{attribute 'linkalways'} 
{attribute 'no_explicit_call' := 'This FB is a CLASS and must be accessed using methods or properties'}
{attribute 'enable_dynamic_creation'}
FUNCTION_BLOCK _ETcVnVectorCompareMethod EXTENDS EnumDatatypeBase
VAR
	localData : ETcVnVectorCompareMethod;
	activeData : REFERENCE TO ETcVnVectorCompareMethod;
	enumBaseDatatype : _DINT(localData);
END_VAR

METHOD PRIVATE AddLocalEnumeration
VAR_INPUT
	Enumeration : T_MAXSTRING;
	Value : ETcVnVectorCompareMethod;
END_VAR
AddEnumeration(Enumeration, Value);
END_METHOD

PROPERTY PUBLIC Address : PVOID
GET
Address := ADR(activeData);
END_GET
END_PROPERTY

METHOD PUBLIC ClearReference
VAR_INPUT
END_VAR
activeData REF= localData;
SetBaseDatatypeReference();
END_METHOD

METHOD PUBLIC Clone : I_Datatype
VAR
    pClone : POINTER TO _ETcVnVectorCompareMethod;
END_VAR
pClone := __NEW(_ETcVnVectorCompareMethod(InitialValue := Value));
Clone := pClone^;
END_METHOD

METHOD FB_init : BOOL
VAR_INPUT
	bInitRetains : BOOL; // if TRUE, the retain variables are initialized (warm start / cold start)
	bInCopyCode : BOOL;  // if TRUE, the instance afterwards gets moved into the copy code (online change)
	InitialValue : ETcVnVectorCompareMethod;
END_VAR
localData := InitialValue;
AddBaseDatatype(enumBaseDatatype);
ClearReference();

AddLocalEnumeration('TCVN_VCM_EUCLIDEAN', ETcVnVectorCompareMethod.TCVN_VCM_EUCLIDEAN);
AddLocalEnumeration('TCVN_VCM_ELEMENTWISE', ETcVnVectorCompareMethod.TCVN_VCM_ELEMENTWISE);
END_METHOD

PROPERTY PUBLIC Identifier : T_MAXSTRING
GET
Identifier := 'ETcVnVectorCompareMethod';
END_GET
END_PROPERTY

METHOD IsEnumeratorValueEqual : BOOL
VAR_INPUT
	Enumerator : I_KeyValueForwardEnumerator;
END_VAR
VAR
	storedValue : ETcVnVectorCompareMethod;
END_VAR
IF NOT Enumerator.TryGet(storedValue) THEN
	RETURN;
END_IF

IsEnumeratorValueEqual := storedValue = activeData;
END_METHOD

METHOD PUBLIC MakeReferenceTo
VAR_INPUT
	ReferenceTarget : REFERENCE TO ETcVnVectorCompareMethod;
END_VAR
activeData REF= ReferenceTarget;
SetBaseDatatypeReference();
END_METHOD

METHOD PROTECTED SetBaseDatatypeReference
VAR_INPUT
END_VAR
enumBaseDatatype.MakeReferenceTo(activeData);
END_METHOD

PROPERTY PUBLIC Size : UDINT
GET
Size := SIZEOF(activeData);
END_GET
END_PROPERTY

METHOD TryMakeReferenceTo : BOOL
VAR_INPUT
	Target : I_Datatype;
END_VAR
VAR
	pTargetData : POINTER TO ETcVnVectorCompareMethod;
END_VAR
IF NOT IsEquivalentTo(Target) THEN
	RETURN;
END_IF

pTargetData := Target.Address;
activeData REF= pTargetData^;
SetBaseDatatypeReference();
TryMakeReferenceTo := TRUE;
END_METHOD

PROPERTY PUBLIC Value : ETcVnVectorCompareMethod
GET
Value := activeData;
END_GET
SET
activeData := Value;
END_SET
END_PROPERTY

END_FUNCTION_BLOCK

(* stored: Version 1.1.0.1, ProductVersion 3.1.4024.13
   POU _ETcVnVectorCompareMethod: Id {03fd922e-608d-0226-20b8-a4f8ac454f24}, SpecialFunc None
   Folder Core: Id {8b8c620e-939d-00e4-0029-f0483bdd4afd}
   Folder Protected: Id {62f7bef5-1c7f-0dde-3fe3-ee3cb2754b3f}
   Folder Customize: Id {2855be75-c159-055c-3312-db7c8260df19}
   Folder Constructor: Id {58b7c4de-e1d9-0980-1098-cda8bf9cd678}
   Folder Private: Id {247d0c3a-806b-0bf6-2d51-5f9e7cfddb0d}
   Folder Protected: Id {0a887545-6216-0086-212f-f1f02c7730c5}
   Method AddLocalEnumeration: Id {e3b2018a-9c21-04de-25f6-2c6ed08d0390}
   Property Address: Id {c9558d60-d6a8-0d39-0170-58529bad7f84}
   Get Get: Id {95751e6b-9ef5-083a-11ef-45d95d5d53bb}
   Method ClearReference: Id {aaafbda6-d1cc-0c51-08c3-f85067a573de}
   Method Clone: Id {1b076b57-c32e-083b-25e0-bfa46519ad07}
   Method FB_init: Id {6873e8be-bcc0-08b0-3f8a-8640f530f080}
   Property Identifier: Id {1b781b04-1297-070a-2576-1beeac5e0eea}
   Get Get: Id {70a539f7-8985-0092-3eb9-b80ac2d40f3e}
   Method IsEnumeratorValueEqual: Id {c3392460-2bfe-0f4d-021c-abd02bec148f}
   Method MakeReferenceTo: Id {30c88ff2-6903-0be5-2956-1037a2ad19c8}
   Method SetBaseDatatypeReference: Id {1f46f972-8aa2-0689-1149-1b744ae70941}
   Property Size: Id {01da506e-4a11-077c-2d29-5acf91a7fbf0}
   Get Get: Id {212b0a50-1aa6-0ba8-2edf-3d1c2e6f0919}
   Method TryMakeReferenceTo: Id {11a4d1b2-7254-08d5-3df9-bfd152c40a57}
   Property Value: Id {2da2b243-c5c9-0c2f-30cf-2bd7c68a1816}
   Get Get: Id {4f52870d-3178-02c1-26b6-fb6da094f75c}
   Set Set: Id {a0fbe4a4-bc76-0aed-273c-89005b3cdb25} *)
